(* CODESYS project codesys-default.export

Project tree, tasks and I/O mapping:
  Advantech_ADAM_5560_WinCE_V3 : Advantech ADAM-5560 WinCE V3, Advantech Co., Ltd., version 3.5.7.10
    application Application
    Backplane : Backplane, Advantech Co., Ltd., version 3.5.7.10
        unmapped channels: System Information, WatchDog
      <Empty>
      <Empty>
      <Empty>
      <Empty>
      <Empty>
      <Empty>
      <Empty>
  Advantech_Control_x86_RTE_V3 : Advantech Control x86 RTE V3, Advantech Co., Ltd., version 3.5.10.0
    application Application
    System_Diagnosis : System Diagnosis, Advantech Co., Ltd., version 3.5.10.0
        unmapped channels: System Information
  Advantech_Control_x86_RTE_V3_x64 : Advantech Control x86 RTE V3 x64, Advantech Co., Ltd., version 3.5.10.0
    application Application
    System_Diagnosis : System Diagnosis, Advantech Co., Ltd., version 3.5.10.0
        unmapped channels: System Information
  Advantech_SoftMotion_x86_RTE_V3 : Advantech SoftMotion x86 RTE V3, Advantech Co., Ltd., version 3.5.10.0
    application Application
    System_Diagnosis : System Diagnosis, Advantech Co., Ltd., version 3.5.10.0
        unmapped channels: System Information
    SoftMotion General Axis Pool
  Advantech_SoftMotion_x86_RTE_V3_x64 : Advantech SoftMotion x86 RTE V3 x64, Advantech Co., Ltd., version 3.5.10.0
    application Application
    System_Diagnosis : System Diagnosis, Advantech Co., Ltd., version 3.5.10.0
        unmapped channels: System Information
    SoftMotion General Axis Pool
  CODESYS_Control_for_PLCnext_SL : CODESYS Control for PLCnext SL, CODESYS, order no. 2302000033, version 4.22.0.0
    application Application
    SoftMotion General Axis Pool
    Axioline : PLCNext Axioline, CODESYS, version 4.22.0.0
  CODESYS_Control_RTE_V3 : CODESYS Control RTE V3, CODESYS, order no. 305017, version 3.5.21.40
    application Application
  CODESYS_Control_RTE_V3_x64 : CODESYS Control RTE V3 x64, CODESYS, version 3.5.21.40
    application Application
  CODESYS_Control_Win_V3 : CODESYS Control Win V3, CODESYS, version 3.5.21.40
    application Application
  Device : CODESYS Control Win V3 x64, CODESYS, version 3.5.21.40
    application Application
      libraries: Standard, 3.5.18.0 (System)
      task MainTask (cyclic, interval t#20ms, priority 1) calls PLC_PRG
      global variables GVL
      program PLC_PRG [ST]
      function block TEST [ST]
*)

// Device/Application/GVL
{attribute 'qualified_only'}
VAR_GLOBAL
END_VAR

// Device/Application/PLC_PRG
PROGRAM PLC_PRG
VAR
END_VAR

END_PROGRAM

// Device/Application/TEST
FUNCTION_BLOCK TEST
VAR_INPUT
END_VAR
VAR_OUTPUT
END_VAR
VAR
END_VAR

END_FUNCTION_BLOCK
